                num_barreno := str_cat("Barreno: ",barrenoActual)
                tcp_actual := get_actual_tcp_pose()
                X_actual := str_cat("     X: ",tcp_actual[0])
                Y_actual := str_cat("     Y: ",tcp_actual[1])
                pos_barreno := str_cat(X_actual,Y_actual)
                Script: textmsg(num_barreno,pos_barreno)
              Poses_taladrado := pose_add(get_actual_tcp_pose(), bajada_broca)
              Waypoint Waypoint (Variable): motionParameters(jointSpeed=1.047198 jointAcceleration=1.396263 cartesianSpeed=0.01 cartesianAcceleration=0.01); variable=Poses_taladrado
              bajada_broca := pose_add(bajada_broca, p[0,0,0.018,0,0,0])
            MoveDirectionNode (selectedDirection=ZPlus toolParams=0.03, 0.04)
              Until DISTANCE (allowActions=false deceleration=3 distanceNodeType=STOP) Distance=0.05; motionParameters(blendRadius=0)
            MoveJ speed 60 deg/s, acceleration 80 deg/s^2 (useActiveTCP=true) feature=Base
              Waypoint Waypoint (Variable): variable=internos
            Wait Sleep waitTime=0.3
            Set DigitalOutput pin=config_out[1]; digitalValue=0
            Wait Sleep waitTime=0.3
            If barrenoActual≟13 or barrenoActual≟27
              MoveDirectionNode (selectedDirection=ZPlus)
                Until DISTANCE (allowActions=false deceleration=3 distanceNodeType=STOP) Distance=0.03; motionParameters(blendRadius=0)
              MoveJ speed 60 deg/s, acceleration 80 deg/s^2 (useActiveTCP=true) feature=Base
                Waypoint Zona_izq1: TCP in base x=721.637 y=-174.262 z=505.425 mm, rx=2.3235 ry=2.1144 rz=0.0001 rad; joints [0.067, -89.734, -90.405, -179.332, -89.71, -0.034] deg
                Waypoint Posicion_Cero: TCP in base x=0.551 y=-324.742 z=1651.532 mm, rx=-0.0041 ry=-0.0154 rz=-3.05 rad; joints [-0.003, -90.003, 0.004, -89.999, -0.001, 0] deg
              Call Quitar_Broca_Chida
              Call Poner_Broca
              MoveJ speed 60 deg/s, acceleration 80 deg/s^2 (useActiveTCP=true) feature=Base
                Waypoint Posicion_Cero: TCP in base x=0.551 y=-324.742 z=1651.532 mm, rx=-0.0041 ry=-0.0154 rz=-3.05 rad; joints [-0.003, -90.003, 0.004, -89.999, -0.001, 0] deg
                Waypoint Zona_izq1: TCP in base x=721.637 y=-174.262 z=505.425 mm, rx=2.3235 ry=2.1144 rz=0.0001 rad; joints [0.067, -89.734, -90.405, -179.332, -89.71, -0.034] deg
            barrenoActual := barrenoActual+1
      Folder Linea 2 a 217
        broca := 217
        Folder Buje_inicial
          Buje_Inicial := L2B2
        Folder Buje_final
          Buje_Final := L2B1
        barrenosTotales := 27
        barrenoActual := 1
        Loop While (checkContinuously=false) expression=barrenoActual≤barrenosTotales
          MoveL speed 250 mm/s, acceleration 1200 mm/s^2 (useActiveTCP=true) feature=Base
            bajada_broca := p[0,0,0.018,0,0,0]
            internos := interpolate_pose(Buje_Inicial, Buje_Final, ((barrenoActual)-1)/((barrenosTotales)-1))
            Folder Alturas
              If barrenoActual≟3 or barrenoActual≟5 or barrenoActual≟7 or barrenoActual≟9 or barrenoActual≟11 or barrenoActual≟13 or barrenoActual≟15 or barrenoActual≟17 or barrenoActual≟19 or barrenoActual≟21 or barrenoActual≟23 or barrenoActual≟25 or barrenoActual≟27 or barrenoActual≟1
                Set ExpressionOutput pin=mensaje_mw10; expression=200
                Wait DigitalInput pin=Continuar_M30; digitalValue=1
                Wait Sleep waitTime=1
                Set ExpressionOutput pin=mensaje_mw10; expression=150
                Wait Sleep waitTime=1
              MoveJ speed 60 deg/s, acceleration 80 deg/s^2 (useActiveTCP=true) feature=Base
                Waypoint Waypoint (Variable): variable=internos
              Wait Sleep waitTime=2
              If P1h[2]<P2h[2]
                acomodin := (altura/(barrenosTotales-1))*(barrenoActual-1)
                tcp_chido := get_actual_tcp_pose()
                offset_bajada := p[tcp_chido[0],tcp_chido[1],((alta-0.0095)-(acomodin/1000)),tcp_chido[3],tcp_chido[4],tcp_chido[5]]
                MoveL speed 15 mm/s, acceleration 30 mm/s^2 (useActiveTCP=true) feature=Base
                  Waypoint Waypoint (Variable): variable=offset_bajada
              Else 
                acomodin := (altura/(barrenosTotales-1))*(26-(barrenoActual-1))
                tcp_chido := get_actual_tcp_pose()
                offset_bajada := p[tcp_chido[0],tcp_chido[1],((alta-0.0095)-(acomodin/1000)),tcp_chido[3],tcp_chido[4],tcp_chido[5]]
                MoveL speed 15 mm/s, acceleration 30 mm/s^2 (useActiveTCP=true) feature=Base
                  Waypoint Waypoint (Variable): variable=offset_bajada
            Folder Freemove
              Wait Sleep waitTime=2
              Script: freedrive_mode()
              Wait Sleep waitTime=2.5
              Script: end_freedrive_mode()
            Wait Sleep waitTime=0.3
            Set DigitalOutput pin=config_out[1]; digitalValue=1
            Wait Sleep waitTime=1
            Wait Sleep waitTime=0.3
            Wait Sleep waitTime=0.3
            Wait Sleep waitTime=0.3
            Loop Counting (count=1) loopVariable(name=Loop_78)
              Poses_taladrado := pose_sub(get_actual_tcp_pose(), bajada_broca)
              Waypoint Waypoint (Variable): motionParameters(jointSpeed=1.047198 jointAcceleration=1.396263 cartesianSpeed=0.001 cartesianAcceleration=0.005); variable=Poses_taladrado
              If bajada_broca≟p[0,0,0.018,0,0,0]
                num_barreno := str_cat("Barreno: ",barrenoActual)
                tcp_actual := get_actual_tcp_pose()
                X_actual := str_cat("     X: ",tcp_actual[0])
                Y_actual := str_cat("     Y: ",tcp_actual[1])
                pos_barreno := str_cat(X_actual,Y_actual)
                Script: textmsg(num_barreno,pos_barreno)
              Poses_taladrado := pose_add(get_actual_tcp_pose(), bajada_broca)
              Waypoint Waypoint (Variable): motionParameters(jointSpeed=1.047198 jointAcceleration=1.396263 cartesianSpeed=0.01 cartesianAcceleration=0.01); variable=Poses_taladrado
              bajada_broca := pose_add(bajada_broca, p[0,0,0.018,0,0,0])
            MoveDirectionNode (selectedDirection=ZPlus toolParams=0.03, 0.04)
              Until DISTANCE (allowActions=false deceleration=3 distanceNodeType=STOP) Distance=0.05; motionParameters(blendRadius=0)
            MoveJ speed 60 deg/s, acceleration 80 deg/s^2 (useActiveTCP=true) feature=Base
              Waypoint Waypoint (Variable): variable=internos
            Wait Sleep waitTime=0.3
            Set DigitalOutput pin=config_out[1]; digitalValue=0
            Wait Sleep waitTime=0.3
            If barrenoActual≟13
              MoveDirectionNode (selectedDirection=ZPlus)
                Until DISTANCE (allowActions=false deceleration=3 distanceNodeType=STOP) Distance=0.03; motionParameters(blendRadius=0)
              MoveJ speed 60 deg/s, acceleration 80 deg/s^2 (useActiveTCP=true) feature=Base
                Waypoint Zona_izq1: TCP in base x=721.637 y=-174.262 z=505.425 mm, rx=2.3235 ry=2.1144 rz=0.0001 rad; joints [0.067, -89.734, -90.405, -179.332, -89.71, -0.034] deg
                Waypoint Posicion_Cero: TCP in base x=0.551 y=-324.742 z=1651.532 mm, rx=-0.0041 ry=-0.0154 rz=-3.05 rad; joints [-0.003, -90.003, 0.004, -89.999, -0.001, 0] deg
              Call Quitar_Broca_Chida
              Call Poner_Broca
              MoveJ speed 60 deg/s, acceleration 80 deg/s^2 (useActiveTCP=true) feature=Base
                Waypoint Posicion_Cero: TCP in base x=0.551 y=-324.742 z=1651.532 mm, rx=-0.0041 ry=-0.0154 rz=-3.05 rad; joints [-0.003, -90.003, 0.004, -89.999, -0.001, 0] deg
                Waypoint Zona_izq1: TCP in base x=721.637 y=-174.262 z=505.425 mm, rx=2.3235 ry=2.1144 rz=0.0001 rad; joints [0.067, -89.734, -90.405, -179.332, -89.71, -0.034] deg
            ElseIf barrenoActual≟27
              MoveDirectionNode (selectedDirection=ZPlus)
                Until DISTANCE (allowActions=false deceleration=3 distanceNodeType=STOP) Distance=0.03; motionParameters(blendRadius=0)
              MoveJ speed 60 deg/s, acceleration 80 deg/s^2 (useActiveTCP=true) feature=Base
                Waypoint Zona_izq1: TCP in base x=721.637 y=-174.262 z=505.425 mm, rx=2.3235 ry=2.1144 rz=0.0001 rad; joints [0.067, -89.734, -90.405, -179.332, -89.71, -0.034] deg
                Waypoint Posicion_Cero: TCP in base x=0.551 y=-324.742 z=1651.532 mm, rx=-0.0041 ry=-0.0154 rz=-3.05 rad; joints [-0.003, -90.003, 0.004, -89.999, -0.001, 0] deg
              Call Quitar_Broca_Chida
              Set DigitalOutput pin=carrusel_home; digitalValue=1
              Wait Sleep waitTime=1
              Set DigitalOutput pin=carrusel_home; digitalValue=0
              Set ExpressionOutput pin=mensaje_mw10; expression=120
              Wait DigitalInput pin=Continuar_M30; digitalValue=1
              Wait Sleep waitTime=1
              Set ExpressionOutput pin=mensaje_mw10; expression=100
              Wait DigitalInput pin=Continuar_M30; digitalValue=1
              Wait Sleep waitTime=1
              MoveJ speed 60 deg/s, acceleration 80 deg/s^2 (useActiveTCP=true) feature=Base
                Waypoint Traslacion_izq: TCP in base x=-174.237 y=-721.63 z=505.386 mm, rx=-3.1292 ry=0.1412 rz=-0.0002 rad; joints [-90, -90.001, -90.002, -180, -90.003, -0.001] deg
            barrenoActual := barrenoActual+1
    SuppressedNode
      Set ExpressionOutput pin=lado_izq_mw9; expression=1
    Folder Traslacion
      MoveJ speed 60 deg/s, acceleration 80 deg/s^2 (useActiveTCP=true) feature=Base
        Waypoint Traslacion_izq: TCP in base x=-174.237 y=-721.63 z=505.386 mm, rx=-3.1292 ry=0.1412 rz=-0.0002 rad; joints [-90, -90.001, -90.002, -180, -90.003, -0.001] deg
      Set ExpressionOutput pin=mensaje_mw10; expression=105
      Wait DigitalInput pin=Continuar_M30; digitalValue=1
      Wait Sleep waitTime=1
      Set ExpressionOutput pin=mensaje_mw10; expression=110
      Wait DigitalInput pin=Continuar_M30; digitalValue=1
      Wait Sleep waitTime=1
      Set DigitalOutput pin=postrnas_m187; digitalValue=1
      Wait Sleep waitTime=1
      Set DigitalOutput pin=Home_M20; digitalValue=1
      Wait Sleep waitTime=1
      Set DigitalOutput pin=Home_M20; digitalValue=0
      Set DigitalOutput pin=postrnas_m187; digitalValue=0
      Wait Sleep waitTime=5
    Folder Apagar
      Set ExpressionOutput pin=mensaje_mw10; expression=115
      Wait DigitalInput pin=Continuar_M30; digitalValue=1
      Wait Sleep waitTime=1
      MoveJ speed 60 deg/s, acceleration 80 deg/s^2 (useActiveTCP=true) feature=Base
        Waypoint Waypoint_9: TCP in base x=-174.329 y=119.284 z=905.669 mm, rx=2.0147 ry=-0.0908 rz=0.0576 rad; joints [-90.002, -15.002, -90.002, -189.996, -89.997, -0.004] deg
        Waypoint Waypoint_8: TCP in base x=-173.7 y=-124.883 z=163.166 mm, rx=3.1302 ry=-0.1403 rz=0.0027 rad; joints [-90.002, -15, -153.998, -189.998, -89.998, -0.004] deg
        Waypoint Off_izquierda: TCP in base x=-173.642 y=-15.442 z=55.621 mm, rx=-1.8394 ry=0.083 rz=0.0614 rad; joints [-89.997, -89.996, -154.003, -190.002, -89.995, 0.005] deg
      Set ExpressionOutput pin=mensaje_mw10; expression=0
      Wait Sleep waitTime=1
      Wait DigitalInput pin=Continuar_M30; digitalValue=1
      Wait Sleep waitTime=1
      Popup Warning (haltProgram=true message=DAS apagado inputType=Text)
  ElseIf Lado_Correr≟2
    Popup Warning (haltProgram=true message=Apagar DAS inputType=Text)
  ElseIf Lado_Correr≟3
    Popup Warning (haltProgram=true message=Apagar DAS inputType=Text)
  Else 
    Lado := False
    Popup Warning (haltProgram=true message=DAS no anclado inputType=Text)
SubProgram -> Poner_Broca
SubProgram -> Quitar_Broca_Chida
SubProgram -> Calibracion
SubProgram Poner_Broca (keepSynchronizedWithDisk=false)
  If Lado_Correr≟1
    Folder Poner_Broca
      Set DigitalOutput pin=ini_cambro_m289; digitalValue=0
      MoveJ speed 60 deg/s, acceleration 80 deg/s^2 (useActiveTCP=true) feature=Base
        Waypoint Precambio_izq: TCP in base x=0.343 y=460.224 z=419.989 mm, rx=0.2109 ry=3.1246 rz=-0.0222 rad; joints [-122.778, -120.749, 120.698, 0.478, 59.722, -0.747] deg
      MoveL speed 250 mm/s, acceleration 1200 mm/s^2 (useActiveTCP=true) feature=Base
        Waypoint Dejar_izq: TCP in base x=0.402 y=460.235 z=60.506 mm, rx=0.2111 ry=3.1246 rz=-0.0221 rad; joints [-122.769, -100.667, 150.148, -49.108, 59.633, -0.646] deg
      Set DigitalOutput pin=ini_cambro_m289; digitalValue=1
      Wait Sleep waitTime=3.8
      Set DigitalOutput pin=ini_cambro_m289; digitalValue=0
      Wait Sleep waitTime=0.5
      Wait DigitalInput pin=fciclocarr_m292; digitalValue=0
      Wait Sleep waitTime=0.5
      Script: freedrive_mode()
      Wait Sleep waitTime=2
      Script: end_freedrive_mode()
      MoveJ speed 60 deg/s, acceleration 80 deg/s^2 (useActiveTCP=true) feature=Base
        Waypoint Dejar_izq: TCP in base x=0.402 y=460.235 z=60.506 mm, rx=0.2111 ry=3.1246 rz=-0.0221 rad; joints [-122.769, -100.667, 150.148, -49.108, 59.633, -0.646] deg
      MoveL speed 250 mm/s, acceleration 1200 mm/s^2 (useActiveTCP=true) feature=Base
        Waypoint Precambio_izq: TCP in base x=0.343 y=460.224 z=419.989 mm, rx=0.2109 ry=3.1246 rz=-0.0222 rad; joints [-122.778, -120.749, 120.698, 0.478, 59.722, -0.747] deg
  ElseIf Lado_Correr≟2
    SuppressedNode
      Popup Message (haltProgram=false message=__ inputType=Text)
  ElseIf Lado_Correr≟3
    SuppressedNode
      Popup Message (haltProgram=false message=__ inputType=Text)
  Else 
    Lado := False
    Popup Warning (haltProgram=true message=DAS no anclado inputType=Text)
SubProgram Quitar_Broca_Chida (keepSynchronizedWithDisk=false)
  If Lado_Correr≟1
    Folder Quitar_Broca
      MoveJ speed 60 deg/s, acceleration 80 deg/s^2 (useActiveTCP=true) feature=Base
        Loop Counting (count=1) loopVariable(name=Loop_3)
          MoveL speed 250 mm/s, acceleration 1200 mm/s^2 (useActiveTCP=true) feature=Base
            MoveJ speed 60 deg/s, acceleration 80 deg/s^2 (useActiveTCP=true) feature=Base
              Waypoint Precambio_izq: TCP in base x=0.343 y=460.224 z=419.989 mm, rx=0.2109 ry=3.1246 rz=-0.0222 rad; joints [-122.778, -120.749, 120.698, 0.478, 59.722, -0.747] deg
            Waypoint Dejar_izq: motionParameters(jointSpeed=1.047198 jointAcceleration=1.396263 cartesianSpeed=0.1 cartesianAcceleration=0.05); TCP in base x=0.402 y=460.235 z=60.506 mm, rx=0.2111 ry=3.1246 rz=-0.0221 rad; joints [-122.769, -100.667, 150.148, -49.108, 59.633, -0.646] deg
            Folder Freemove
              Wait Sleep waitTime=2
              Script: freedrive_mode()
              Wait Sleep waitTime=2.5
              Script: end_freedrive_mode()
            Set DigitalOutput pin=outputbroc_m291; digitalValue=1
            Wait Sleep waitTime=0.5
            Set DigitalOutput pin=outputbroc_m291; digitalValue=0
            Wait Sleep waitTime=0.5
            Wait DigitalInput pin=fciclocarr_m292; digitalValue=0
            Wait Sleep waitTime=0.5
            Folder Freemove
              Wait Sleep waitTime=0.5
              Script: freedrive_mode()
              Wait Sleep waitTime=2.5
              Script: end_freedrive_mode()
            Waypoint Precambio_izq: TCP in base x=0.343 y=460.224 z=419.989 mm, rx=0.2109 ry=3.1246 rz=-0.0222 rad; joints [-122.778, -120.749, 120.698, 0.478, 59.722, -0.747] deg
            Set DigitalOutput pin=avancarrusel_m7; digitalValue=1
            Wait Sleep waitTime=1.1
            Set DigitalOutput pin=avancarrusel_m7; digitalValue=0
  ElseIf Lado_Correr≟2
    SuppressedNode
      Popup Message (haltProgram=false message=_____ inputType=Text)
  ElseIf Lado_Correr≟3
    SuppressedNode
      Popup Message (haltProgram=false message=_____ inputType=Text)
  Else 
    Lado := False
    Popup Warning (haltProgram=true message=DAS no anclado inputType=Text)
SubProgram Calibracion (keepSynchronizedWithDisk=false)
  Folder Offsets factor
    SuppressedNode
      broca := 1645
    L1B1x := ((0.09523476)/(0.09525))*(0.09523476)
    L1B1y := ((-0.01278382)/(-0.0127))*(-0.01278382)
    L1B2x := ((0.75575414)/(0.75565))*(0.75575414)
    L1B2y := ((-0.01279398)/(-0.0127))*(-0.01279398)
    L2B1x := ((0.09675299)/(0.09525))*(0.09675299)
    L2B1y := ((0.3937)/(0.3937))*(0.3937)
    L2B2x := ((0.757306777)/(0.75565))*(0.757306777)
    L2B2y := ((0.393684081)/(0.3937))*(0.393684081)
  If Lado_Correr≟1
    Folder Subvariables
      muestras := 1
      muestrasTomadas := 0
      P1 := p[0,0,0,0,0,0]
      P2 := p[0,0,0,0,0,0]
      P3 := p[0,0,0,0,0,0]
      P4 := p[0,0,0,0,0,0]
      P1h := p[0,0,0,0,0,0]
      P2h := p[0,0,0,0,0,0]
      altura := 0
      rotaciones := p[0,0,0,0,0,0]
      PosFinal := p[0,0,0,0,0,0]
      m1 := 0
      m2 := 0
      b1 := 0
      b2 := 0
      Xd := 0
      Yd := 0
      Xp := 0
      Yp := 0
      Xfin := 0
      Yfin := 0
    Folder Calibracion
      MoveL speed 250 mm/s, acceleration 1200 mm/s^2 (useActiveTCP=true) feature=Base
        MoveDirectionNode (selectedDirection=ZPlus)
          Until DISTANCE (allowActions=false deceleration=3 distanceNodeType=STOP) Distance=0.1; motionParameters(blendRadius=0)
        MoveJ speed 60 deg/s, acceleration 80 deg/s^2 (useActiveTCP=true) feature=Base
          Waypoint Zona_izq1: TCP in base x=721.637 y=-174.262 z=505.425 mm, rx=2.3235 ry=2.1144 rz=0.0001 rad; joints [0.067, -89.734, -90.405, -179.332, -89.71, -0.034] deg
        MoveL speed 250 mm/s, acceleration 1200 mm/s^2 (useActiveTCP=true) feature=Base
          MoveJ speed 60 deg/s, acceleration 80 deg/s^2 (useActiveTCP=true) feature=Base
            If pos_eje7_mw13≟2
              Waypoint Paso1_Izq1: TCP in base x=724.517 y=-11.189 z=99.711 mm, rx=-2.3926 ry=-2.0358 rz=0 rad; joints [17.663, -102.285, -121.211, -135.887, -68.394, -0.223] deg
            ElseIf pos_eje7_mw13≟3
              Waypoint Paso1_Izq2: TCP in base x=724.528 y=34.912 z=88.856 mm, rx=-2.3926 ry=-2.0359 rz=-0.0001 rad; joints [22.207, -103.255, -121.439, -134.653, -63.855, -0.278] deg
          Folder P1
            Loop While (checkContinuously=false) expression=muestrasTomadas<muestras
              MoveJ speed 60 deg/s, acceleration 80 deg/s^2 (useActiveTCP=true) feature=Base
                If pos_eje7_mw13≟2
                  Waypoint Sacar1_izq1: TCP in base x=394.634 y=-44.739 z=37.51 mm, rx=-2.3926 ry=-2.0358 rz=-0.0001 rad; joints [37.23, -71.258, -158.634, -129.28, -48.851, -0.528] deg
                ElseIf pos_eje7_mw13≟3
                  Waypoint Sacar1_izq2: TCP in base x=389.881 y=-27.806 z=38.705 mm, rx=2.392 ry=2.0358 rz=0.0009 rad; joints [42.726, -69.346, -159.321, -130.335, -43.368, -0.703] deg
              Wait Sleep waitTime=0.5
              MoveDirectionNode (selectedDirection=YMinus toolParams=0.0013, 2.0E-4)
                Until TOOL_CONTACT_DETECTION (allowActions=false retraction=0 decelerationAcceleration=9 decelerationAngularAcceleration=34.906585)
              Wait Sleep waitTime=2
              P1 := pose_add(get_actual_tcp_pose(), P1)
              muestrasTomadas := muestrasTomadas+1
            muestrasTomadas := 0
            var_1 := (P1[0])/muestras
            var_2 := (P1[1])/muestras
            rotaciones := get_actual_tcp_pose()
            var_3 := rotaciones[3]
            var_4 := rotaciones[4]
            var_5 := rotaciones[5]
            P1 := p[var_1,var_2,-0.37,var_3,var_4,var_5]
          Folder P1h
            Loop While (checkContinuously=false) expression=muestrasTomadas<muestras
              MoveDirectionNode (selectedDirection=YPlus)
                Until DISTANCE (allowActions=false deceleration=3 distanceNodeType=STOP) Distance=0.04; motionParameters(blendRadius=0)
              MoveJ speed 60 deg/s, acceleration 80 deg/s^2 (useActiveTCP=true) feature=Base
                If pos_eje7_mw13≟2
                  Waypoint Sacar1h_izq1: TCP in base x=464.657 y=-49.256 z=69.987 mm, rx=-2.3927 ry=-2.0358 rz=0.0001 rad; joints [26.501, -78.699, -149.376, -131.231, -59.572, -0.353] deg
                ElseIf pos_eje7_mw13≟3
                  Waypoint Sacar1h_izq2: TCP in base x=461.503 y=-33.306 z=40.342 mm, rx=2.392 ry=2.0358 rz=0.001 rad; joints [29.936, -82.374, -151.482, -125.363, -56.168, -0.42] deg
              Wait Sleep waitTime=0.5
              MoveDirectionNode (selectedDirection=ZMinus toolParams=0.0013, 2.0E-4)
                Until TOOL_CONTACT_DETECTION (allowActions=false retraction=0 decelerationAcceleration=9 decelerationAngularAcceleration=34.906585)
              Wait Sleep waitTime=2
              P1h := pose_add(get_actual_tcp_pose(), P1h)
              muestrasTomadas := muestrasTomadas+1
            muestrasTomadas := 0
            var_1 := (P1h[0])/muestras
            var_2 := (P1h[1])/muestras
            var_9 := (P1h[2])/muestras
            rotaciones := get_actual_tcp_pose()
            var_3 := rotaciones[3]
            var_4 := rotaciones[4]
            var_5 := rotaciones[5]
            P1h := p[var_1,var_2,var_9,var_3,var_4,var_5]
          MoveJ speed 60 deg/s, acceleration 80 deg/s^2 (useActiveTCP=true) feature=Base
            If pos_eje7_mw13≟2
              Waypoint Paso1_Izq1: TCP in base x=724.517 y=-11.189 z=99.711 mm, rx=-2.3926 ry=-2.0358 rz=0 rad; joints [17.663, -102.285, -121.211, -135.887, -68.394, -0.223] deg
            ElseIf pos_eje7_mw13≟3
              Waypoint Paso1_Izq2: TCP in base x=724.528 y=34.912 z=88.856 mm, rx=-2.3926 ry=-2.0359 rz=-0.0001 rad; joints [22.207, -103.255, -121.439, -134.653, -63.855, -0.278] deg
          Folder P2
            Loop While (checkContinuously=false) expression=muestrasTomadas<muestras
              MoveJ speed 60 deg/s, acceleration 80 deg/s^2 (useActiveTCP=true) feature=Base
                If pos_eje7_mw13≟2
                  Waypoint Sacar2_izq1: TCP in base x=1149.582 y=-41.957 z=41.791 mm, rx=-2.3927 ry=-2.0358 rz=-0.0002 rad; joints [8.25, -139.784, -65.969, -153.677, -77.737, -0.116] deg
                ElseIf pos_eje7_mw13≟3
                  Waypoint Sacar2_izq2: TCP in base x=1142.673 y=-24.562 z=46.993 mm, rx=2.3926 ry=2.0359 rz=0.0001 rad; joints [9.318, -138.87, -67.13, -153.424, -76.675, -0.132] deg
              Wait Sleep waitTime=0.5
              MoveDirectionNode (selectedDirection=YMinus toolParams=0.0013, 2.0E-4)
                Until TOOL_CONTACT_DETECTION (allowActions=false retraction=0 decelerationAcceleration=9 decelerationAngularAcceleration=34.906585)
              Wait Sleep waitTime=2
              P2 := pose_add(get_actual_tcp_pose(), P2)
              muestrasTomadas := muestrasTomadas+1
            muestrasTomadas := 0
            var_1 := (P2[0])/muestras
            var_2 := (P2[1])/muestras
            rotaciones := get_actual_tcp_pose()
            var_3 := rotaciones[3]
            var_4 := rotaciones[4]
            var_5 := rotaciones[5]
            P2 := p[var_1,var_2,-0.37,var_3,var_4,var_5]
          MoveJ speed 60 deg/s, acceleration 80 deg/s^2 (useActiveTCP=true) feature=Base
            If pos_eje7_mw13≟2
              Waypoint Paso1_Izq1: TCP in base x=724.517 y=-11.189 z=99.711 mm, rx=-2.3926 ry=-2.0358 rz=0 rad; joints [17.663, -102.285, -121.211, -135.887, -68.394, -0.223] deg
            ElseIf pos_eje7_mw13≟3
              Waypoint Paso1_Izq2: TCP in base x=724.528 y=34.912 z=88.856 mm, rx=-2.3926 ry=-2.0359 rz=-0.0001 rad; joints [22.207, -103.255, -121.439, -134.653, -63.855, -0.278] deg
          Folder P2h
            Loop While (checkContinuously=false) expression=muestrasTomadas<muestras
              MoveJ speed 60 deg/s, acceleration 80 deg/s^2 (useActiveTCP=true) feature=Base
                If pos_eje7_mw13≟2
                  Waypoint Sacar2h_izq1: TCP in base x=1124.539 y=-46.74 z=50.049 mm, rx=-2.3926 ry=-2.0358 rz=-0.0001 rad; joints [8.182, -137.133, -70.07, -152.232, -77.814, -0.114] deg
                ElseIf pos_eje7_mw13≟3
                  Waypoint Sacar2h_izq2: TCP in base x=1123.4 y=-32.87 z=50.433 mm, rx=-2.3926 ry=-2.0358 rz=-0.0001 rad; joints [9.014, -136.974, -70.324, -152.132, -76.982, -0.124] deg
              Wait Sleep waitTime=0.5
              MoveDirectionNode (selectedDirection=ZMinus toolParams=0.0013, 2.0E-4)
                Until TOOL_CONTACT_DETECTION (allowActions=false retraction=0 decelerationAcceleration=9 decelerationAngularAcceleration=34.906585)
              Wait Sleep waitTime=2
              P2h := pose_add(get_actual_tcp_pose(), P2h)
              muestrasTomadas := muestrasTomadas+1
            muestrasTomadas := 0
            var_1 := (P2h[0])/muestras
            var_2 := (P2h[1])/muestras
            var_9 := (P2h[2])/muestras
            rotaciones := get_actual_tcp_pose()
            var_3 := rotaciones[3]
            var_4 := rotaciones[4]
            var_5 := rotaciones[5]
            P2h := p[var_1,var_2,var_9,var_3,var_4,var_5]
          MoveJ speed 60 deg/s, acceleration 80 deg/s^2 (useActiveTCP=true) feature=Base
            If pos_eje7_mw13≟2
              Waypoint Paso1_Izq1: TCP in base x=724.517 y=-11.189 z=99.711 mm, rx=-2.3926 ry=-2.0358 rz=0 rad; joints [17.663, -102.285, -121.211, -135.887, -68.394, -0.223] deg
            ElseIf pos_eje7_mw13≟3
              Waypoint Paso1_Izq2: TCP in base x=724.528 y=34.912 z=88.856 mm, rx=-2.3926 ry=-2.0359 rz=-0.0001 rad; joints [22.207, -103.255, -121.439, -134.653, -63.855, -0.278] deg
          Folder m1
            var_1 := (P1[0])
            var_2 := (P1[1])
            var_3 := (P2[0])
            var_4 := (P2[1])
            m1 := (var_4-var_2)/(var_3-var_1)
          Folder b1
            b1 := ((m1*var_1)-var_2)*(-1)
          MoveJ speed 60 deg/s, acceleration 80 deg/s^2 (useActiveTCP=true) feature=Base
            Waypoint Paso2_izq1: TCP in base x=414.118 y=-280.673 z=89.978 mm, rx=-2.3928 ry=-2.0356 rz=0 rad; joints [-18.236, -84.335, -142.099, -133.065, -104.295, 0.11] deg
          Folder P3
            Loop While (checkContinuously=false) expression=muestrasTomadas<muestras
              MoveJ speed 60 deg/s, acceleration 80 deg/s^2 (useActiveTCP=true) feature=Base
                If pos_eje7_mw13≟2
                  Waypoint Sacar3_izq1: TCP in base x=375.457 y=-406.999 z=39.986 mm, rx=-2.3929 ry=-2.0356 rz=0 rad; joints [-38.01, -97.791, -136.069, -125.593, -124.076, 0.332] deg
                ElseIf pos_eje7_mw13≟3
                  Waypoint Sacar3_izq2: TCP in base x=371.851 y=-391.262 z=39.216 mm, rx=-2.3927 ry=-2.0355 rz=0 rad; joints [-36.577, -96.531, -137.746, -125.188, -122.647, 0.319] deg
              Wait Sleep waitTime=0.5
              MoveDirectionNode (selectedDirection=XMinus toolParams=0.0013, 2.0E-4)
                Until TOOL_CONTACT_DETECTION (allowActions=false retraction=0 decelerationAcceleration=9 decelerationAngularAcceleration=34.906585)
              Wait Sleep waitTime=2
              P3 := pose_add(get_actual_tcp_pose(), P3)
              muestrasTomadas := muestrasTomadas+1
            muestrasTomadas := 0
            var_1 := (P3[0])/muestras
            var_2 := (P3[1])/muestras
            rotaciones := get_actual_tcp_pose()
            var_3 := rotaciones[3]
            var_4 := rotaciones[4]
            var_5 := rotaciones[5]
            P3 := p[var_1,var_2,-0.37,var_3,var_4,var_5]
          MoveJ speed 60 deg/s, acceleration 80 deg/s^2 (useActiveTCP=true) feature=Base
            Waypoint Paso2_izq1: TCP in base x=414.118 y=-280.673 z=89.978 mm, rx=-2.3928 ry=-2.0356 rz=0 rad; joints [-18.236, -84.335, -142.099, -133.065, -104.295, 0.11] deg
          Folder P4
            Loop While (checkContinuously=false) expression=muestrasTomadas<muestras
              MoveJ speed 60 deg/s, acceleration 80 deg/s^2 (useActiveTCP=true) feature=Base
                If pos_eje7_mw13≟2
                  Waypoint Sacar4_izq1: TCP in base x=373.966 y=-146.95 z=39.429 mm, rx=-2.3929 ry=-2.0356 rz=0 rad; joints [10.396, -74.338, -156.788, -128.296, -75.672, -0.159] deg
                ElseIf pos_eje7_mw13≟3
                  Waypoint Sacar4_izq2: TCP in base x=370.43 y=-132.19 z=39.809 mm, rx=-2.3928 ry=-2.0356 rz=-0.0001 rad; joints [15.041, -72.036, -157.906, -129.449, -71.029, -0.21] deg
              Wait Sleep waitTime=0.5
              MoveDirectionNode (selectedDirection=XMinus toolParams=0.0013, 2.0E-4)
                Until TOOL_CONTACT_DETECTION (allowActions=false retraction=0 decelerationAcceleration=9 decelerationAngularAcceleration=34.906585)
              Wait Sleep waitTime=2
              P4 := pose_add(get_actual_tcp_pose(), P4)
              muestrasTomadas := muestrasTomadas+1
            muestrasTomadas := 0
            var_1 := (P4[0])/muestras
            var_2 := (P4[1])/muestras
            rotaciones := get_actual_tcp_pose()
            var_3 := rotaciones[3]
            var_4 := rotaciones[4]
            var_5 := rotaciones[5]
            P4 := p[var_1,var_2,-0.37,var_3,var_4,var_5]
          MoveJ speed 60 deg/s, acceleration 80 deg/s^2 (useActiveTCP=true) feature=Base
            Waypoint Paso2_izq1: TCP in base x=414.118 y=-280.673 z=89.978 mm, rx=-2.3928 ry=-2.0356 rz=0 rad; joints [-18.236, -84.335, -142.099, -133.065, -104.295, 0.11] deg
          Folder m2
            var_1 := (P3[0])
            var_2 := (P3[1])
            var_3 := (P4[0])
            var_4 := (P4[1])
            m2 := (var_4-var_2)/(var_3-var_1)
          Folder b2
            b2 := ((m2*var_1)-var_2)*(-1)
          Folder Xd y Yd
            Xd := (b2-b1)/(m1-m2)
            Yd := (m1*Xd)+b1
          SuppressedNode
            Folder Zp
              var_10 := (pow((P1h[0]-P2h[0]), 2))+(pow((P1h[1]-P2h[1]), 2))
              var_11 := (pow((P1h[2]-P2h[2]), 2))+(var_10)
              var_12 := sqrt(var_10/var_11)
          Folder Xp y Yp
            Xp := ((1)/(sqrt((m1*m1)+1)))*(1)
            Yp := ((m2)/(sqrt((m2*m2)+1)))*(1)
          Folder Origen
            Xfin := (((0*(-1)*Xp)-(Xd)-(0*(1/m2)))*(-1))*(1)
            Yfin := (((0*(-1)*Yp)-(Yd)+(0*(-1)*m1))*(-1))*(1)
            rotaciones := get_actual_tcp_pose()
            var_3 := rotaciones[3]
            var_4 := rotaciones[4]
            var_5 := rotaciones[5]
            If broca≟1645
              PosFinal := p[Xfin-0.00208915,Yfin-0.00208915,0.420,var_3,var_4,var_5]
            ElseIf broca≟1935
              PosFinal := p[Xfin-0.00245745,Yfin-0.00245745,0.420,var_3,var_4,var_5]
            ElseIf broca≟217
              PosFinal := p[Xfin-0.0027559,Yfin-0.0027559,0.420,var_3,var_4,var_5]
            origen := PosFinal
          Folder Linea1_Buje1
            Xfin := ((((L1B1x)*(-1)*Xp)-(Xd)-((L1B1y)*(1/m2)))*(-1))*(1)
            Yfin := ((((L1B1y)*(-1)*Yp)-(Yd)+((L1B1x)*(-1)*m1))*(-1))*(1)
            rotaciones := get_actual_tcp_pose()
            var_3 := rotaciones[3]
            var_4 := rotaciones[4]
            var_5 := rotaciones[5]
            If broca≟1645
              PosFinal := p[(Xfin-0.00208915)*1000,(Yfin-0.00208915)*1000,0.420,var_3,var_4,var_5]
            ElseIf broca≟1935
              PosFinal := p[Xfin-0.00245745,Yfin-0.00245745,0.420,var_3,var_4,var_5]
            ElseIf broca≟217
              PosFinal := p[Xfin-0.0027559,Yfin-0.0027559,0.420,var_3,var_4,var_5]
            Linea1_Buje1 := PosFinal
          Folder Linea1_Buje27
            Xfin := ((((L1B2x)*(-1)*Xp)-(Xd)-((L1B2y)*(1/m2)))*(-1))*(1)
            Yfin := ((((L1B2y)*(-1)*Yp)-(Yd)+((L1B2x)*(-1)*m1))*(-1))*(1)
            rotaciones := get_actual_tcp_pose()
            var_3 := rotaciones[3]
            var_4 := rotaciones[4]
            var_5 := rotaciones[5]
            If broca≟1645
              PosFinal := p[(Xfin-0.00208915)*1000,(Yfin-0.00208915)*1000,0.420,var_3,var_4,var_5]
            ElseIf broca≟1935
              PosFinal := p[Xfin-0.00245745,Yfin-0.00245745,0.420,var_3,var_4,var_5]
            ElseIf broca≟217
              PosFinal := p[Xfin-0.0027559,Yfin-0.0027559,0.420,var_3,var_4,var_5]
            Linea1_Buje27 := PosFinal
          Folder Linea2_Buje1
            Xfin := ((((L2B1x)*(-1)*Xp)-(Xd)-((L2B1y)*(1/m2)))*(-1))*(1)
            Yfin := ((((L2B1y)*(-1)*Yp)-(Yd)+((L2B1x)*(-1)*m1))*(-1))*(1)
            rotaciones := get_actual_tcp_pose()
            var_3 := rotaciones[3]
            var_4 := rotaciones[4]
            var_5 := rotaciones[5]
            If broca≟1645
              PosFinal := p[(Xfin-0.00208915)*1000,(Yfin-0.00208915)*1000,0.420,var_3,var_4,var_5]
            ElseIf broca≟1935
              PosFinal := p[Xfin-0.00245745,Yfin-0.00245745,0.420,var_3,var_4,var_5]
            ElseIf broca≟217
              PosFinal := p[Xfin-0.0027559,Yfin-0.0027559,0.420,var_3,var_4,var_5]
            Linea2_Buje1 := PosFinal
          Folder Linea2_Buje27
            Xfin := ((((L2B2x)*(-1)*Xp)-(Xd)-((L2B2y)*(1/m2)))*(-1))*(1)
            Yfin := ((((L2B2y)*(-1)*Yp)-(Yd)+((L2B2x)*(-1)*m1))*(-1))*(1)
            rotaciones := get_actual_tcp_pose()
            var_3 := rotaciones[3]
            var_4 := rotaciones[4]
            var_5 := rotaciones[5]
            If broca≟1645
              PosFinal := p[(Xfin-0.00208915)*1000,(Yfin-0.00208915)*1000,0.420,var_3,var_4,var_5]
            ElseIf broca≟1935
              PosFinal := p[Xfin-0.00245745,Yfin-0.00245745,0.420,var_3,var_4,var_5]
            ElseIf broca≟217
              PosFinal := p[Xfin-0.0027559,Yfin-0.0027559,0.420,var_3,var_4,var_5]
            Linea2_Buje27 := PosFinal
          Folder Altura
            If P1h[2]<P2h[2]
              altura := (P2h[2]-P1h[2])*1000
              alta := P2h[2]
            Else 
              altura := (P1h[2]-P2h[2])*1000
              alta := P1h[2]
          MoveDirectionNode (selectedDirection=ZPlus)
            Until DISTANCE (allowActions=false deceleration=3 distanceNodeType=STOP) Distance=0.1; motionParameters(blendRadius=0)
          MoveJ speed 60 deg/s, acceleration 80 deg/s^2 (useActiveTCP=true) feature=Base
            Waypoint Zona_izq1: TCP in base x=721.637 y=-174.262 z=505.425 mm, rx=2.3235 ry=2.1144 rz=0.0001 rad; joints [0.067, -89.734, -90.405, -179.332, -89.71, -0.034] deg
  ElseIf Lado_Correr≟2
    SuppressedNode
      Popup Message (haltProgram=false message=__ inputType=Text)
  ElseIf Lado_Correr≟3
    SuppressedNode
      Popup Message (haltProgram=false message=__ inputType=Text)
  Else 
    Lado := False
    Popup Warning (haltProgram=true message=DAS no anclado inputType=Text)
